FUNCTION_BLOCK DM_CLT (* Remote Device Management Client *)
  (* Standard: 61499 Demo ITA; Function: Device Management; Description: Client for Remote Device Management - Use with CLIENT_2_1 *)
  (* Version 0.4, 2002-01-01, JHC, Rockwell Automation, Added WAIT, request_timeout. *)
  (* Version 0.3, 2001-01-21, JHC, Rockwell Automation, Changed to ServiceManager interface *)
  (* Version 0.2, 2001-01-14, JHC, Rockwell Automation, Changed event inputs *)
  (* Version 0.1, 2001-01-04, JHC, Rockwell Automation, Added STATUS input *)
  (* Version 0.0, 2000-12-31, JHC, Rockwell Automation, Initial version *)
  (* Compiler header: package fb.rt; *)
  (* Compiler Java IBM VisualAge 3.0 *)
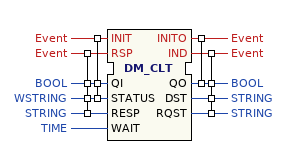
  EVENT_INPUT
    INIT WITH QI, STATUS; (* Comm Client Initialization Response *)
    RSP WITH QI, STATUS, RESP; (* Remote Management Response *)
  END_EVENT
  EVENT_OUTPUT
    INITO WITH QO; (* Initialize/Terminate Comm Client *)
    IND WITH QO, DST, RQST; (* Remote Management Request to Comm Client *)
  END_EVENT
  VAR_INPUT
    QI : BOOL; (* Event Input Qualifier *)
    STATUS : WSTRING; (* Communications Status *)
    RESP : STRING; (* XML-encoded Response *)
    WAIT : TIME := t#2s; (* Request Timeout Period(Maximum allowed IND/RSP Delay) *)
  END_VAR
  VAR_OUTPUT
    QO : BOOL; (* Event Output Qualifier *)
    DST : STRING; (* Destination for RQST *)
    RQST : STRING; (* XML-encoded Request *)
  END_VAR
  SERVICE DM_CLT/SystemManager
    SEQUENCE connect
      SystemManager.connect() -> DM_CLT.INITO+();
      DM_CLT.INIT+() -> SystemManager.connected();
    END_SEQUENCE
    SEQUENCE connect_err
      SystemManager.connect() -> DM_CLT.INITO+();
      DM_CLT.INIT-(STATUS) -> SystemManager.error(STATUS);
    END_SEQUENCE
    SEQUENCE normal_request
      SystemManager.request(DST,RQST) -> DM_CLT.IND+(DST,RQST);
      DM_CLT.RSP+(RESP) -> SystemManager.response(RESP);
    END_SEQUENCE
    SEQUENCE request_comm_err
      SystemManager.request(DST,RQST) -> DM_CLT.IND+(DST,RQST);
      DM_CLT.RSP-(STATUS) -> SystemManager.error(STATUS);
    END_SEQUENCE
    SEQUENCE request_timeout (* No RSP within DT after IND *)
      SystemManager.request(DST,RQST) -> DM_CLT.IND+(DST,RQST);
      -> SystemManager.error(STATUS="NOT_READY");
    END_SEQUENCE
    SEQUENCE disconnect
      SystemManager.disconnect() -> DM_CLT.INITO-();
      DM_CLT.INIT-(STATUS) -> SystemManager.disconnected(STATUS);
    END_SEQUENCE
  END_SERVICE
END_FUNCTION_BLOCK
